KUKA KRL data list: art_statistics.dat

&ACCESS RV2
&REL 4
&PARAM DISKPATH = KRC:\R1\TP\ART
DEFDAT  art_statistics PUBLIC
; Count.
DECL GLOBAL INT ARTStatContainerCount[2]
ARTStatContainerCount[1]=292
ARTStatContainerCount[2]=313
DECL GLOBAL INT ARTStatContInBatch[2]
ARTStatContInBatch[1]=204
ARTStatContInBatch[2]=259
DECL GLOBAL INT ARTStatProductCount=17632
DECL GLOBAL INT ARTStatFailsCount=0
; Speed.
DECL GLOBAL REAL ARTStatSpeedInProduct=2.36589479
DECL GLOBAL REAL ARTStatSpeedInContainer=0.0812325105
; Fail rate. FailRate = Fails / Product
DECL GLOBAL INT ARTStatFailRate=0

DECL GLOBAL REAL ARTStatRunTime=7453.81641
DECL GLOBAL REAL ARTStatWaitTime=0.0
DECL GLOBAL REAL ARTStatErrorTime=338.428162

DECL GLOBAL CONST INT DEF_STAT_TIMER_WAIT=20
DECL GLOBAL CONST INT DEF_STAT_TIMER_ERR=21
DECL GLOBAL CONST INT DEF_STAT_TIMER_RUN=22

DECL GLOBAL CONST INT ART_ProdPerCycle=2
DECL GLOBAL CONST INT ART_ContainerPerCycle=1

DECL GLOBAL BOOL ARTStatisticsResetCmd=FALSE

ENDDAT
